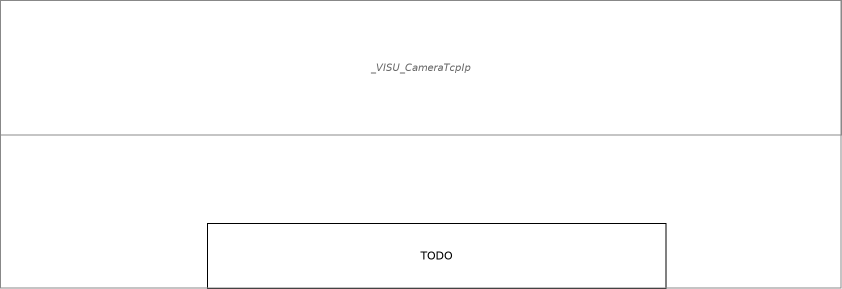
VISUALIZATION _VISU_SystronCamera  // 842x289
    Rectangle (207,223 459x66), "TODO"
    Frame (0,0 842x135)
        shows _VISU_CameraTcpIp(m_Inst := PRG_PRINT.fbLineCamera)
END_VISUALIZATION

(* stored: Version 1.1.0.1, ProductVersion 3.1.4024.3
   Visu _VISU_SystronCamera: Id {03102516-653a-4736-9bd1-25f7bbb0545e} *)
